SUBAPPLICATION GreenWhiteBackground_Zusammenklappen (* Subapplication Type *)
  (* Standard: 61499-2 *)
  (* Version 1.0, 2023-02-11, franz *)
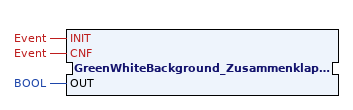
  EVENT_INPUT
    INIT;
    CNF;
  END_EVENT
  VAR_INPUT
    OUT : BOOL;
  END_VAR
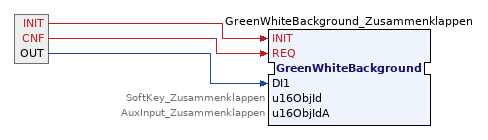
  SUBAPPS
    GreenWhiteBackground_Zusammenklappen : GreenWhiteBackground(u16ObjId := SoftKey_Zusammenklappen, u16ObjIdA := AuxInput_Zusammenklappen);
  END_SUBAPPS
  EVENT_CONNECTIONS
    INIT TO GreenWhiteBackground_Zusammenklappen.INIT;
    CNF TO GreenWhiteBackground_Zusammenklappen.REQ;
  END_CONNECTIONS
  DATA_CONNECTIONS
    OUT TO GreenWhiteBackground_Zusammenklappen.DI1;
  END_CONNECTIONS
END_SUBAPPLICATION
